// TwinCAT 3 PLC project Doble_Gato_PLC
// ProgramVersion: 3.1.4023.0
// libraries:
//   Tc2_Standard, * (Beckhoff Automation GmbH)
//   Tc2_System, * (Beckhoff Automation GmbH)
//   Tc2_Utilities, * (Beckhoff Automation GmbH)
//   Tc3_EventLogger, * (Beckhoff Automation GmbH)
//   Tc3_Module, * (Beckhoff Automation GmbH)
// project tree:
//   DUTs/ eBeltObject.TcDUT, eFeed.TcDUT, BeltStatus.TcDUT, OUTPUT_LABELS.TcDUT, INPUT_LABELS.TcDUT, U_IN_IO_Translate.TcDUT, U_OUT_IO_Translate.TcDUT
//   FBs/ FB_ButtonBox.TcPOU, FB_GatoPerro.TcPOU, FB_BeltControl.TcPOU
//   F/ F_TemperatureMethod.TcPOU
//   GVLs/ GENERAL.TcGVL
//   GVLs/IO/ IN.TcGVL, OUT.TcGVL
//   GVLs/SAFETY/ SAFETY.TcGVL
//   / PlcTask.TcTTO, SlowTask.TcTTO
//   POUs/ OVERVIEW_FBD.TcPOU, MAIN.TcPOU, P_Temperature_Obs.TcPOU, P_BACKGROUND.TcPOU, P_SAFETY.TcPOU, README.TcPOU
//   POUs/GENERAL/ P_WritePersistentData.TcPOU
// real-time tasks:
//   TASK PlcTask: cycle T#10ms, priority 20, ADS port 350
//   TASK SlowTask: cycle T#50000us, priority 30, ADS port 351
// I/O:
//   DEVICE Device 3 (EtherCAT Automation Protocol), AmsNetId 5.62.144.216.4.1
//   DEVICE Device 1 (EtherCAT), AmsNetId 5.62.144.216.2.1
//     Term 1 (EK1200) [EK1200-5000 EtherCAT Power supply (2A E-Bus)]
//       Term 2 (EL3204) [EL3204 4Ch. Ana. Input PT100 (RTD)]
//       Term 3 (EL1008) [EL1008 8Ch. Dig. Input 24V, 3ms]
//       Term 4 (EL2008) [EL2008 8Ch. Dig. Output 24V, 0.5A]
//       Term 5 (EL1809) [EL1809 16Ch. Dig. Input 24V, 3ms]
//       Term 6 (EL2809) [EL2809 16Ch. Dig. Output 24V, 0.5A]
//       Term 7 (EK1122) [EK1122 2 port EtherCAT junction]
//         Term 8 (EK1100) [EK1100 EtherCAT Coupler (2A E-Bus)]
//           Term 9 (EL1008) [EL1008 8Ch. Dig. Input 24V, 3ms]
//           Term 10 (EL2008) [EL2008 8Ch. Dig. Output 24V, 0.5A]
//           Term 11 (EL9011) [EL9011 End Terminal]
// variable links:
//   Doble Gato PLC/Doble Gato PLC Instance <-> Device 1 (EtherCAT)
//     SlowTask Inputs/GENERAL.EthercatDevState <-> Inputs/DevState
//     SlowTask Outputs/GENERAL.EthercatDevCtrl <-> Outputs/DevCtrl
//   Doble Gato PLC/Doble Gato PLC Instance <-> Device 1 (EtherCAT)/Term 1 (EK1200)/Term 2 (EL3204)
//     SlowTask Inputs/IN.ANALOG[{1..4}] <-> RTD Inputs Channel {1..4}/Value  (4 links)
//   Doble Gato PLC/Doble Gato PLC Instance <-> Device 1 (EtherCAT)/Term 1 (EK1200)/Term 3 (EL1008)
//     PlcTask Inputs/IN._DI/bArray[{1..8}] <-> Channel {1..8}/Input  (8 links)
//   Doble Gato PLC/Doble Gato PLC Instance <-> Device 1 (EtherCAT)/Term 1 (EK1200)/Term 4 (EL2008)
//     PlcTask Outputs/OUT._DO/bArray[{1..8}] <-> Channel {1..8}/Output  (8 links)
//   Doble Gato PLC/Doble Gato PLC Instance <-> Device 1 (EtherCAT)/Term 1 (EK1200)/Term 5 (EL1809)
//     PlcTask Inputs/IN._DI/bArray[{9..24}] <-> Channel {1..16}/Input  (16 links)
//   Doble Gato PLC/Doble Gato PLC Instance <-> Device 1 (EtherCAT)/Term 1 (EK1200)/Term 6 (EL2809)
//     PlcTask Outputs/OUT._DO/bArray[{9..24}] <-> Channel {1..16}/Output  (16 links)
//   Doble Gato PLC/Doble Gato PLC Instance <-> Device 1 (EtherCAT)/Term 1 (EK1200)/Term 7 (EK1122)/Term 8 (EK1100)/Term 10 (EL2008)
//     PlcTask Outputs/OUT._DO/bArray[{25..32}] <-> Channel {1..8}/Output  (8 links)
//   Doble Gato PLC/Doble Gato PLC Instance <-> Device 1 (EtherCAT)/Term 1 (EK1200)/Term 7 (EK1122)/Term 8 (EK1100)/Term 9 (EL1008)
//     PlcTask Inputs/IN._DI/bArray[{25..32}] <-> Channel {1..8}/Input  (8 links)
//   Doble Gato PLC/Doble Gato PLC Instance <-> Device 3 (EtherCAT Automation Protocol)
//     SlowTask Inputs/GENERAL.EthercatDev1 <-> Inputs/DevState

CONFIGURATION Doble_Gato_PLC
    RESOURCE PLC ON TwinCAT3
        TASK PlcTask(INTERVAL := T#10ms, PRIORITY := 20);
        TASK SlowTask(INTERVAL := T#50000us, PRIORITY := 30);
        PROGRAM MAIN WITH PlcTask : MAIN;
        PROGRAM P_Temperature_Obs WITH SlowTask : P_Temperature_Obs;
    END_RESOURCE
END_CONFIGURATION

// ---- DUTs/eBeltObject.TcDUT
{attribute 'qualified_only'}
{attribute 'strict'}
TYPE eBeltObject :
(
	EMPTY := 0,
	GATO := 1,
	PERRO := 2,
	MAGIC := 3
);
END_TYPE

// ---- DUTs/eFeed.TcDUT
{attribute 'qualified_only'}
{attribute 'to_string'}
TYPE eFeed :
(
	Stop := 0,
	Ready,
	Running,
	Fault,
	State4
);
END_TYPE

// ---- DUTs/BeltStatus.TcDUT
{attribute 'qualified_only'}
{attribute 'strict'}
TYPE BeltStatus :
(
	Idle := 0,
	Ready,
	Running,
	Error_status := 100

);
END_TYPE

// ---- DUTs/OUTPUT_LABELS.TcDUT
TYPE OUTPUT_LABELS :
STRUCT
//===== 	Box EL2008			
ButtonBox_Light	:		BOOL;
bOutput2		:		BOOL;
bOutput3		:		BOOL;
bOutput4		:		BOOL;
bOutput5		:		BOOL;
bOutput6		:		BOOL;
bOutput7		:		BOOL;
DoorSensor_Activator		:		BOOL;
//===== 	Box EL2809
bOutput9		:		BOOL;
bOutput10		:		BOOL;
bOutput11		:		BOOL;
bOutput12		:		BOOL;
bOutput13		:		BOOL;
bOutput14		:		BOOL;
bOutput15		:		BOOL;
bOutput16		:		BOOL;
bOutput17		:		BOOL;
bOutput18		:		BOOL;
bOutput19		:		BOOL;
bOutput20		:		BOOL;
bOutput21		:		BOOL;
bOutput22		:		BOOL;
bOutput23		:		BOOL;
bOutput24		:		BOOL;
//===== 	EK1100 EL2008
VFD_RUN_14			:		BOOL;
VFD_BACKWARD_15		:		BOOL;
VFD_FORWARD_16		:		BOOL;
LIGHT_White		:		BOOL;
LIGHT_Green		:		BOOL;
bOutput30		:		BOOL;
bOutput31		:		BOOL;
bOutput32		:		BOOL;

END_STRUCT
END_TYPE

// ---- DUTs/INPUT_LABELS.TcDUT
TYPE INPUT_LABELS :
STRUCT
//===== 	Box EL1008			
BTN_Feed		:		BOOL;
SWITCH_Right		:		BOOL;
SWITCH_Left		:		BOOL;
bInput4		:		BOOL;
bInput5		:		BOOL;
bInput6		:		BOOL;
bInput7		:		BOOL;
SM_Door_Sensor1		:		BOOL;
//===== 	Box EL1809
bInput9		:		BOOL;
SM_Wheel_RotationCount		:		BOOL;
bInput11		:		BOOL;
SL_Wheel_LightSensor1		:		BOOL;
bInput13		:		BOOL;
bInput14		:		BOOL;
bInput15		:		BOOL;
bInput16		:		BOOL;
bInput17		:		BOOL;
bInput18		:		BOOL;
bInput19		:		BOOL;
bInput20		:		BOOL;
bInput21		:		BOOL;
bInput22		:		BOOL;
bInput23		:		BOOL;
bInput24		:		BOOL;
//====		EL1100 -> EL1008
VFD_READY_20		:		BOOL;
bInput26		:		BOOL;
VFD_24		:		BOOL;
bInput28		:		BOOL;
VFD_26		:		BOOL;
bInput30		:		BOOL;
bInput31		:		BOOL;
SM_Gato_MagnetSensor		:		BOOL;

END_STRUCT
END_TYPE

// ---- DUTs/U_IN_IO_Translate.TcDUT
TYPE U_IN_IO_Translate :
UNION
	bArray :	ARRAY[1..32] OF BOOL;
	_Label :		INPUT_LABELS;
END_UNION
END_TYPE

// ---- DUTs/U_OUT_IO_Translate.TcDUT
TYPE U_OUT_IO_Translate :
UNION
	bArray :	ARRAY[1..32] OF BOOL;
	_Label :		OUTPUT_LABELS;
END_UNION
END_TYPE

// ---- GVLs/GENERAL.TcGVL
{attribute 'qualified_only'}
VAR_GLOBAL
	ReadyForAction		: BOOL;
	BlinkOn				: BOOL;
	BlinkFAST_On		: BOOL;
	BlinkSpecial_On		: BOOL;	
	Motor_OK			: BOOL;
	Manual				: BOOL;
	Auto				: BOOL;

// General information	
	sCelsius: STRING(16);
	sFahrenheit: STRING(16);
	sCosine: STRING(16);
	sKelvin: STRING(16);

	Gato : BOOL;
	Perro : BOOL;
	GatoCount: UINT;
	PerroCount: UINT;	
	
// Linked 'useless' variables to IO
	EthercatDevState 	AT%I*: UINT;
	Term2DevState 		AT%I*: UINT;
	EthercatDevCtrl 	AT%Q*: UINT;
	EthercatDev1		AT%I*: UINT;
	EthercatDev3		AT%I*: UINT;


END_VAR

// ---- GVLs/IO/IN.TcGVL
{attribute 'qualified_only'}
VAR_GLOBAL
	_DI				AT %I*: 	U_IN_IO_Translate;
	ANALOG			AT %I*:		ARRAY[1..4] OF INT;	// Temperature module
	
END_VAR

// ---- GVLs/IO/OUT.TcGVL
{attribute 'qualified_only'}
VAR_GLOBAL
	_DO 			AT%Q*:		U_OUT_IO_Translate;

END_VAR

// ---- GVLs/SAFETY/SAFETY.TcGVL
{attribute 'qualified_only'}
VAR_GLOBAL
	//Turvapiirien tilatiedot
	Safety_OK							AT%Q*	:BOOL;	//
	Doors_OK							AT%Q*	:BOOL;	//
	E_STOP_OK							AT%Q*	:BOOL;	//
	
END_VAR

// ---- POUs/MAIN.TcPOU
PROGRAM MAIN
VAR
	
END_VAR


P_Safety();						// Check doors, safety switches etc. before going through with main program

IF GENERAL.ReadyForAction AND SAFETY.Safety_OK THEN 	// If both signals indicating readyness are given, go through with main tasks.
		P_BACKGROUND();					// Background routines. Blinks etc
		P_WritePersistentData();		// Writes persistent variables to memory every 10 seconds
		OVERVIEW_FBD();					// FBD View of all FB's. Useful visualization of whats happening
			// P_Environment_Control 		-> Is a separate slow task, not to be called from MAIN
END_IF

END_PROGRAM

// ---- POUs/P_SAFETY.TcPOU
PROGRAM P_SAFETY
VAR
	Door1_Box	: BOOL;
	Door2_Fence : BOOL;
	Door3_Workbench : BOOL;
	
END_VAR


A_Doors();	// Checking if doors are open
A_Checks(); // Acting on sensor inputs

	//Virtual switches waiting for physical ones
	SAFETY.E_STOP_OK 		:= TRUE;
	GENERAL.Motor_OK		:= TRUE;
	
//============
// If VFD is ready and Security is satisfactory, global "Good To Go"-signal is given
IF GENERAL.Motor_OK AND SAFETY.Safety_OK THEN
	GENERAL.ReadyForAction := TRUE;
END_IF

ACTION A_Checks:
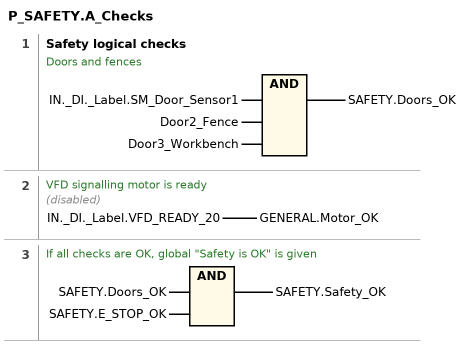
// NETWORK 1: Safety logical checks
// Doors and fences
SAFETY.Doors_OK := IN._DI._Label.SM_Door_Sensor1 AND Door2_Fence AND Door3_Workbench;

// NETWORK 2 (disabled)
// VFD signalling motor is ready
// GENERAL.Motor_OK := IN._DI._Label.VFD_READY_20;

// NETWORK 3
// If all checks are OK, global "Safety is OK" is given
SAFETY.Safety_OK := SAFETY.Doors_OK AND SAFETY.E_STOP_OK;
END_ACTION

ACTION A_Doors:
//"Door sensor" is active Output running to magnet sensor in door
OUT._DO._Label.DoorSensor_Activator := TRUE;

//========================

Door1_Box 		:= IN._DI._Label.SM_Door_Sensor1;	// Previously activated door sensor output is listened here
Door2_Fence 	:= TRUE;							// Not implemented physically	
Door3_Workbench := TRUE;							// Not implemented physically

IF (Door1_Box AND Door2_Fence AND Door3_Workbench) = TRUE THEN	// Checking through all doors and fences
	SAFETY.Doors_OK := TRUE;
	ELSE
		SAFETY.Doors_OK := FALSE;
END_IF
END_ACTION

END_PROGRAM

// ---- POUs/P_BACKGROUND.TcPOU
PROGRAM P_BACKGROUND
VAR
	bDoors : BOOL;
	State: INT;
	
	
//================	
	// Blink timer
	TIME_ON 			: TIME := T#1S;
	TIME_OFF 			: TIME := T#1S;	
	TIME_FAST_ON 		: TIME := T#250MS;
	TIME_FAST_OFF 		: TIME := T#250MS;
	TIME_SPECIAL_ON 	: TIME := T#50MS;
	TIME_SPECIAL_OFF 	: TIME := T#50MS;	
	
	BlinkTimer_ON: TON;
	BlinkTimer_OFF: TON;
	BlinkTimer_FAST_ON: TON;
	BlinkTimer_FAST_OFF: TON;
	BlinkTimer_SPEC_ON: TON;
	BlinkTimer_SPEC_OFF: TON;
	T_ON : BOOL;
	T_OFF : BOOL := TRUE;	
	T_FAST_ON : BOOL;
	T_FAST_OFF : BOOL := TRUE;	
	T_SPEC_ON : BOOL;
	T_SPEC_OFF : BOOL := TRUE;
//==================

	StateSpecial: INT;
	i: INT;
	Input1_RTRIG: R_TRIG;
	Input2_RTRIG: R_TRIG;
	tempCounter: INT;
	tempCounter2: INT;
	bSwitchToggle: BOOL;
END_VAR


//	A_ButtonBoxes();
//	A_FeedButton();
	Blink();
	Blink_Faster();
	Blink_Special();

ACTION A_Beacons:

END_ACTION

ACTION Blink:

BlinkTimer_ON(IN:= T_ON , PT:= TIME_ON , Q=> , ET=> );
IF BlinkTimer_ON.Q THEN
	T_ON 	:= GENERAL.BlinkOn:= FALSE;
	T_OFF 	:= TRUE;	
END_IF

BlinkTimer_OFF(IN:= T_OFF , PT:= TIME_OFF , Q=> , ET=> );
IF BlinkTimer_OFF.Q THEN
	T_ON 	:= GENERAL.BlinkOn := TRUE;
	T_OFF	:= FALSE;
END_IF
END_ACTION

ACTION Blink_Faster:


BlinkTimer_FAST_ON(IN:= T_FAST_ON , PT:= TIME_FAST_ON , Q=> , ET=> );
IF BlinkTimer_FAST_ON.Q THEN
	T_FAST_ON	:= GENERAL.BlinkFAST_On:= FALSE;
	T_FAST_OFF 	:= TRUE;	
END_IF

BlinkTimer_FAST_OFF(IN:= T_FAST_OFF , PT:= TIME_FAST_OFF , Q=> , ET=> );
IF BlinkTimer_FAST_OFF.Q THEN
	T_FAST_ON 	:= GENERAL.BlinkFAST_On := TRUE;
	T_FAST_OFF	:= FALSE;
END_IF
END_ACTION

ACTION Blink_Special:

CASE StateSpecial OF
0:

	IF i > 5 THEN
		StateSpecial := 1;
		i := 0;
		ELSE
		BlinkTimer_SPEC_ON(IN:= T_SPEC_ON , PT:= (TIME_SPECIAL_ON*5) , Q=> , ET=> );
		IF BlinkTimer_SPEC_ON.Q THEN
			T_SPEC_ON 	:= GENERAL.BlinkSpecial_ON:= FALSE;
			T_SPEC_OFF 	:= TRUE;	
		END_IF
		
		BlinkTimer_SPEC_OFF(IN:= T_SPEC_OFF , PT:= (TIME_SPECIAL_OFF*5) , Q=> , ET=> );
		IF BlinkTimer_SPEC_OFF.Q THEN
			T_SPEC_ON 	:= GENERAL.BlinkSpecial_ON := TRUE;
			T_SPEC_OFF	:= FALSE;
		i:= i+1;
		END_IF
	END_IF

	1: 

	IF i > 1 THEN
		StateSpecial := 0;
		i := 0;
		ELSE
		BlinkTimer_SPEC_ON(IN:= T_SPEC_ON , PT:= (TIME_SPECIAL_ON*10) , Q=> , ET=> );
		IF BlinkTimer_SPEC_ON.Q THEN
			T_SPEC_ON 	:= GENERAL.BlinkSpecial_ON:= FALSE;
			T_SPEC_OFF 	:= TRUE;	
		END_IF
		
		BlinkTimer_SPEC_OFF(IN:= T_SPEC_OFF , PT:= (TIME_SPECIAL_OFF*10) , Q=> , ET=> );
		IF BlinkTimer_SPEC_OFF.Q THEN
			T_SPEC_ON 	:= GENERAL.BlinkSpecial_ON := TRUE;
			T_SPEC_OFF	:= FALSE;
			i:= i+1;
		END_IF
	END_IF
END_CASE
END_ACTION

END_PROGRAM

// ---- POUs/GENERAL/P_WritePersistentData.TcPOU
PROGRAM P_WritePersistentData
VAR
	fbWritePersistentData: FB_WritePersistentData;
	StartTON: TON;
	iCounter: INT;

END_VAR

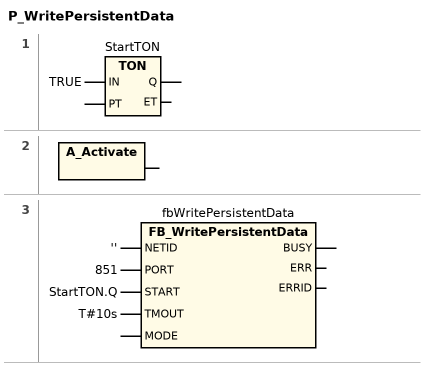
// NETWORK 1
StartTON(IN := TRUE); // TON

// NETWORK 2
A_Activate();

// NETWORK 3
fbWritePersistentData(NETID := '', PORT := 851, START := StartTON.Q, TMOUT := T#10s); // FB_WritePersistentData

ACTION A_Activate:

IF StartTON.Q THEN
	StartTON(IN := FALSE, PT:= T#1M);
		IF NOT fbWritePersistentData.BUSY THEN
		StartTON(IN := TRUE);
		iCounter := iCounter +1; IF iCounter > 50 THEN iCounter := 0; END_IF
		END_IF
END_IF
END_ACTION

END_PROGRAM

// ---- POUs/OVERVIEW_FBD.TcPOU
PROGRAM OVERVIEW_FBD
VAR
	fbButtonBox: FB_ButtonBox;
	fbBeltControl: FB_BeltControl;
	fbGatoPerro: FB_GatoPerro;
END_VAR

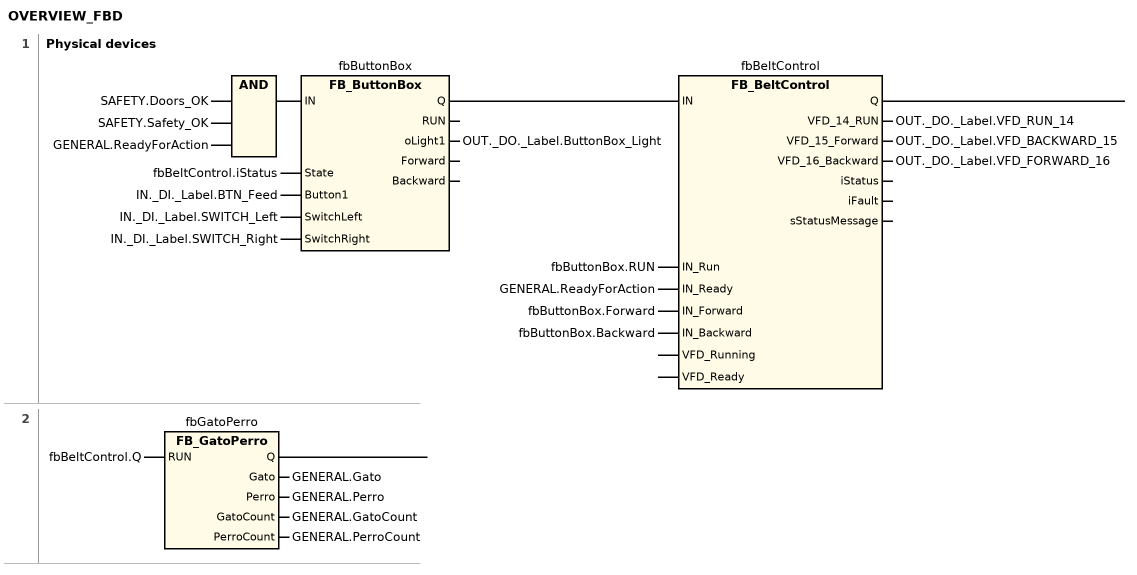
// NETWORK 1: Physical devices
fbButtonBox(
    IN := SAFETY.Doors_OK AND SAFETY.Safety_OK AND GENERAL.ReadyForAction,
    State := fbBeltControl.iStatus,
    Button1 := IN._DI._Label.BTN_Feed,
    SwitchLeft := IN._DI._Label.SWITCH_Left,
    SwitchRight := IN._DI._Label.SWITCH_Right,
    oLight1 => OUT._DO._Label.ButtonBox_Light); // FB_ButtonBox
fbBeltControl(
    IN := fbButtonBox.Q,
    IN_Run := fbButtonBox.RUN,
    IN_Ready := GENERAL.ReadyForAction,
    IN_Forward := fbButtonBox.Forward,
    IN_Backward := fbButtonBox.Backward,
    VFD_14_RUN => OUT._DO._Label.VFD_RUN_14,
    VFD_15_Forward => OUT._DO._Label.VFD_BACKWARD_15,
    VFD_16_Backward => OUT._DO._Label.VFD_FORWARD_16); // FB_BeltControl

// NETWORK 2
fbGatoPerro(
    RUN := fbBeltControl.Q,
    Gato => GENERAL.Gato,
    Perro => GENERAL.Perro,
    GatoCount => GENERAL.GatoCount,
    PerroCount => GENERAL.PerroCount); // FB_GatoPerro

END_PROGRAM

// ---- FBs/FB_ButtonBox.TcPOU
FUNCTION_BLOCK FB_ButtonBox
VAR_INPUT
	IN			: BOOL;
	State : 	(NOT_READY, ALL_READY, RUNNING, STOP, ERROR);	//Local ENUM
	Button1		: BOOL;
	SwitchLeft 	: BOOL;
	SwitchRight : BOOL;
END_VAR
VAR_OUTPUT
	Q 		: BOOL;
	RUN		: BOOL;
	oLight1 : BOOL;	
	Forward 	: BOOL;
	Backward 	: BOOL;
END_VAR
VAR
	BTN_Feed_TRIG: BOOL;
	Rtrig2: R_TRIG;
	Rtrig3: R_TRIG;
	tempCount1: INT;
	tempCount2: INT;
	tempCount3: INT;
	tempCount0: INT;

	RS1: RS;
	SwitchLeftRight_RS: BOOL;
	rTrig1: R_TRIG;
	RS_2: RS;
END_VAR

Q := IN;

// Button press handling
A_InputHandling();

// Button box light controls dictated by the state of Belt Control.
CASE State OF		// State is an input of 1-5 from BeltControl FB
	
	NOT_READY:
		oLight1 := FALSE;

	ALL_READY:
		oLight1 := GENERAL.BlinkOn;
		
	RUNNING:
		oLight1 := TRUE;		
		
	STOP:
		oLight1 := GENERAL.BlinkSpecial_On;

	ERROR:
		oLight1 := GENERAL.BlinkSpecial_On;
		
END_CASE

ACTION A_InputHandling:
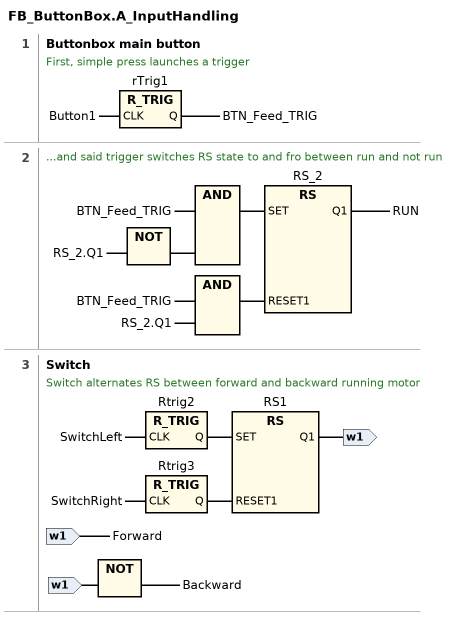
// NETWORK 1: Buttonbox main button
// First, simple press launches a trigger
rTrig1(CLK := Button1); // R_TRIG
BTN_Feed_TRIG := rTrig1.Q;

// NETWORK 2
// ...and said trigger switches RS state to and fro between run and not run
RS_2(SET := BTN_Feed_TRIG AND NOT RS_2.Q1, RESET1 := BTN_Feed_TRIG AND RS_2.Q1); // RS
RUN := RS_2.Q1;

// NETWORK 3: Switch
// Switch alternates RS between forward and backward running motor
Rtrig2(CLK := SwitchLeft); // R_TRIG
Rtrig3(CLK := SwitchRight); // R_TRIG
RS1(SET := Rtrig2.Q, RESET1 := Rtrig3.Q); // RS
Forward := RS1.Q1;
Backward := NOT RS1.Q1;
END_ACTION

END_FUNCTION_BLOCK

// ---- FBs/FB_BeltControl.TcPOU
FUNCTION_BLOCK FB_BeltControl
VAR_INPUT
	IN				: BOOL;
	IN_Run 			: BOOL; // Order to start running
	IN_Ready			: BOOL; // Safety ok, system ok, doors ok
	IN_Forward 			: BOOL;
	IN_Backward			: BOOL;
	VFD_Running		: BOOL;
	VFD_Ready		: BOOL;
	
END_VAR
VAR_OUTPUT
	Q : BOOL;
	VFD_14_RUN 	: BOOL;
	VFD_15_Forward		: BOOL;
	VFD_16_Backward		: BOOL;
	iStatus		: INT;
	iFault		: INT;
	sStatusMessage	: STRING;
END_VAR
VAR
	nMotorState: (NOT_READY, ALL_READY, RUNNING, STOP, ERROR);	//Local ENUM
	Stopping_TON: TON;
	sDirCase: (FORWARD, BACKWARD);
	Frw_Bck: INT;
	fbTcMessage: FB_TcMessage;	//Eventlogger messaging
		bIsInitialized : BOOL;
		bSendMessage : BOOL;
	
	iTempCounter: INT;
END_VAR

M_VariableChanges();
IF NOT IN_Ready THEN		// VFD signal of readiness. Simple way to work safely with VFD
	nMotorState :=0;
END_IF

CASE nMotorState OF
	NOT_READY:	
	sStatusMessage := 'Not ready. Stopped';
		IF IN_Ready THEN
		nMotorState := 1;	// When VFD signals it is ready, we can proceed
		END_IF

	ALL_READY:
	sStatusMessage := 'Ready to run. Motor Stopped';
		VFD_14_RUN := FALSE;
		VFD_15_Forward := FALSE;
		VFD_16_Backward := TRUE;
	
		IF IN_Run THEN		// Inputted signal from buttonbox or other remote to start
			nMotorState := 2;	// Move on to Running-state

			//Also send informational Eventlogger message:
			bIsInitialized := TRUE;
				IF bIsInitialized THEN
					bIsInitialized := FALSE;
					bSendMessage := TRUE;
					fbTcMessage.CreateEx(TC_Events.GatoPerroEvents.Start, 0);
				END_IF
			
		END_IF
		
	RUNNING:
							// Motor can either run forward or backward according to buttonbox switch
		CASE sDirCase  OF			
			BACKWARD:
				VFD_14_RUN := FALSE;
				VFD_15_Forward := TRUE;
				VFD_16_Backward := FALSE;
				sStatusMessage := 'Motor running: Backward';

			FORWARD:
				VFD_14_RUN := TRUE;
				VFD_15_Forward := FALSE;
				VFD_16_Backward := TRUE;
				sStatusMessage := 'Motor running: Forward';
		END_CASE

		IF NOT IN_Run THEN	
			nMotorState := 3;
		END_IF

	STOP:
		sStatusMessage := 'Stopping...';	// Motor is gradually stopped and slight delay is included before new start can be ordered
		VFD_14_RUN := FALSE;
		VFD_15_Forward := FALSE;
		VFD_16_Backward := TRUE;
		
		Stopping_TON(IN:=TRUE , PT:=T#2S , Q=> , ET=> );
			IF Stopping_TON.Q THEN
				Stopping_TON(IN:=FALSE);
				nMotorState := 0;
			END_IF
		
	ERROR:
		sStatusMessage := 'Error state';
	
		
END_CASE

A_Messaging();

ACTION A_Messaging:

//Sends tc eventlogger messages if it is primed previously

IF bSendMessage THEN
	bSendMessage := FALSE;
	iTempCounter := iTempCounter +1;
	fbTcMessage.Send(0);	// 0 = current timestamp
END_IF
END_ACTION

METHOD M_VariableChanges : BOOL
VAR_INPUT
END_VAR

IN 					:= Q;
VFD_15_Forward 		:= IN_Forward;
VFD_16_Backward 	:= IN_Backward;
iStatus 			:= nMotorState;
iFault 				:= 0;
Frw_Bck 			:= BOOL_TO_INT( IN_Forward);
sDirCase		 	:= Frw_Bck;
END_METHOD

END_FUNCTION_BLOCK

// ---- FBs/FB_GatoPerro.TcPOU
FUNCTION_BLOCK FB_GatoPerro
VAR_INPUT
	RUN 		: BOOL;
END_VAR
VAR_OUTPUT
	Q			: BOOL;
	Gato 		: BOOL;
	Perro 		: BOOL;
	GatoCount 	: UINT;
	PerroCount 	: UINT;

END_VAR
VAR
	R_TRIG_0: R_TRIG;
	R_TRIG_1: R_trig;
	GatoTrigger: BOOL;
	WheelLightTrigger: BOOL;
	R_TRIG_2: R_TRIG;
	RotationTrigger: BOOL;
	RotationCount: UINT;
	ObjectCount: UINT;
	GatoPrime: BOOL;
	bGato_or_Perro: BOOL;
	TON_PrimeDelay: TON;
	WheelTime1: TIME;
	WheelTime3: TIME;
	WheelTime2: TIME;
	GP_Check: UINT;
	//A_RotationMeasure VARs	
		tTimeNow: TIME;
		tRotationTime: TIME;
		tTimeStop: TIME;
		iRotations_In_Minute: DWORD;
		iTimenow: DWORD;
		iOneMinute: DWORD;
		iRotationTime: DWORD;
		iOne_Fourth_Rotations_Time: DWORD;
		iTenth_Of_Rotations_Time: DWORD;
		tOne_Fourth_Rotations_Time: TIME;
		tTenth_Of_Rotations_Time: TIME;
	tonLightSDelay: TON;
	ObjectDetectionTime: TIME := T#50MS;
	Prime_Start: BOOL;
END_VAR

Q := RUN;
A_SensorHandling();

// Rotation counter
IF RotationTrigger THEN
	RotationCount := RotationCount +1;

	// We need slight delay before Priming Gato. Perro could be just nearing the Light sensor and register as Gato
	// Lets calculate rotations per minute, divide it to 3/4th rotation and use these later on to prime Gato just in time
	A_RotationMeasure();
		tRotationTime;			// Informational
		iRotations_In_Minute;	// Informational		
END_IF

// Magnet sensor sees Gato
	// Lets add slight delay to avoid mixing with other object on wheel
	TON_PrimeDelay(IN:= Prime_Start, PT:= tOne_Fourth_Rotations_Time, Q=> , ET=> );
		IF GatoTrigger THEN
			Prime_Start := TRUE;
		END_IF
	// When timer is done, Gato is primed and will register in light sensor
		IF TON_PrimeDelay.Q THEN
			GatoPrime := TRUE;
			Prime_Start := FALSE;
		END_IF

// Light sensor sees an object
IF WheelLightTrigger THEN
	ObjectCount := ObjectCount +1;
	IF NOT GatoPrime THEN			// IF Gato is not primed, its Perro
		PerroCount := PerroCount +1;
		bGato_or_Perro := FALSE;
	ELSE							// If Gato is primed in previous steps, its Gato
		GatoPrime := FALSE;
		GatoCount := GatoCount +1;
		bGato_or_Perro := TRUE;
	END_IF

END_IF

// Which one was it
Gato 	:= bGato_or_Perro;
Perro 	:= NOT bGato_or_Perro;
// Finally, lit up a light for whichever object it was
A_SignalLights();

ACTION A_RotationMeasure:
// Calculate RPM from RotationTime, divide it to 1/4th rotation
// Also 1/10th rotation to filter light sensor input
// If rotation time is slowing too much, or stops, reset to 0.2s


// How long does one rotation take
	tTimeNow := TIME();
	tRotationTime := tTimeNow - tTimeStop;
	tTimeStop := tTimeNow;

//Some conversions:
	iTimenow := TIME_TO_DWORD(tTimeNow);
	iOneMinute := TIME_TO_DWORD(T#1M);
	iRotationTime := TIME_TO_DWORD(tRotationTime);

// Rotations_In_Minute
iRotations_In_Minute :=
	iOneMinute/iRotationTime;
	
// 1/4 and 1/10th rotation times
tOne_Fourth_Rotations_Time := DWORD_TO_TIME( iOne_Fourth_Rotations_Time :=
	iRotationTime/4);
tTenth_Of_Rotations_Time := DWORD_TO_TIME( iTenth_Of_Rotations_Time :=
	iRotationTime/10);
END_ACTION

ACTION A_SensorHandling:
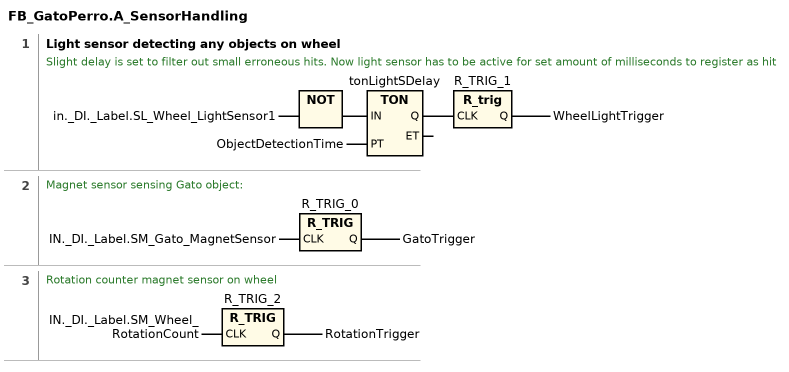
// NETWORK 1: Light sensor detecting any objects on wheel
// Slight delay is set to filter out small erroneous hits. Now light sensor has to be active for set amount of milliseconds to register as hit
tonLightSDelay(IN := NOT in._DI._Label.SL_Wheel_LightSensor1, PT := ObjectDetectionTime); // TON
R_TRIG_1(CLK := tonLightSDelay.Q); // R_trig
WheelLightTrigger := R_TRIG_1.Q;

// NETWORK 2
// Magnet sensor sensing Gato object:
R_TRIG_0(CLK := IN._DI._Label.SM_Gato_MagnetSensor); // R_TRIG
GatoTrigger := R_TRIG_0.Q;

// NETWORK 3
// Rotation counter magnet sensor on wheel
R_TRIG_2(CLK := IN._DI._Label.SM_Wheel_RotationCount); // R_TRIG
RotationTrigger := R_TRIG_2.Q;
END_ACTION

ACTION A_SignalLights:
// Lights signalling which object passed sensor
OUT._DO._Label.LIGHT_White := Gato;
OUT._DO._Label.LIGHT_Green := Perro;
END_ACTION

END_FUNCTION_BLOCK

// ---- POUs/P_Temperature_Obs.TcPOU
PROGRAM P_Temperature_Obs
VAR
	SA_BoxTemperature: REAL;
	rCelsius: REAL;

	rFahrenheit: REAL;
	rKelvin: REAL;
	rCosine: REAL;

END_VAR

// Analogue Temperature sensor inside box
SA_BoxTemperature := IN.ANALOG[1];
//=======================================

//Presenting conversions to display in HMI
F_TemperatureMethod(
	InputTemperature:= SA_BoxTemperature, 
	Celsius=> rCelsius, 
	Fahrenheit=> rFahrenheit, 
	Kelvin=> rKelvin,
	Cosine => rCosine);

// Turning temperature Reals to Global strings.
GENERAL.sCelsius := LREAL_TO_FMTSTR(in:= rCelsius, iPrecision:= 2, bRound:= 1);
GENERAL.sFahrenheit := LREAL_TO_FMTSTR(in:= rFahrenheit, iPrecision:= 2, bRound:= 1);
GENERAL.sKelvin := LREAL_TO_FMTSTR(in:= rKelvin, iPrecision:= 2, bRound:= 1);
GENERAL.sCosine := LREAL_TO_FMTSTR(in:= rCosine, iPrecision:= 5, bRound:= 1);

END_PROGRAM

// ---- F/F_TemperatureMethod.TcPOU
FUNCTION F_TemperatureMethod : REAL
VAR_INPUT
	InputTemperature:	REAL;
END_VAR
VAR_OUTPUT
	Celsius : 		REAL;
	Fahrenheit : 	REAL;
	Kelvin : 		REAL;
	Cosine :		REAL;
END_VAR
VAR
	K: REAL;
	C: REAL;
	F: REAL;
END_VAR

// Function handling analog temperature measurement 
C := InputTemperature/10; 
K := C + 273.15;
F := C * 1.8 +32;

Cosine		 	:= COS(C);
Celsius 		:= C;
Fahrenheit 		:= F;
Kelvin 			:= K;

END_FUNCTION

// ---- POUs/README.TcPOU
PROGRAM README
VAR
END_VAR

(*
//============
NAMING INPUTS USING UNION:
	Give Inputs/Outputs Specific Labels In: 
		DUT/INPUT_LABELS
		DUT/OUTPUT_LABELS
	
	Thus inputs have clear names and address:  
		IN._I._Label.Door_Sensor1
		
	IO is received into Array, and every input is then given a specific Label through Union. 
	IO can still be referenced in array form:
		IN._I.bArray[1];
	Because DUT/Union simply slaps a label on top of bArray[1..32], Door_Sensor1 and bArray[8] are the same thing and thus activate simultaneously.

//============
GATO E PERRO 
	Original idea of this demo project is to showcase and test different inputs, outputs and controls of PLC. Some features are needlessly complicated 
	considering the task, but are used for learning purposes. Several components are scavenged and repurposed, thus giving a but amateurish
	and hacky look to the project, but I still made an effort for professional finish.	

	Name is in Spanish to clearly distinguish test project from actual customer project. Future database names et al continue the same namoing
	convention to make it easier to copy/paste and change variables and names.
	
	End result of project is a cat figure running from dog figure, with magnetic and light sensor observing them.
	Distinguishing cat from a dog can be achieved in many ways, and I chose a middle ground between practicality, budget and reliability.
	Cat figure has a magnet glued behind it, thus "priming" the light sensor 
	-> next time a figure passes light sensor, its a cat. 
	-> If light sensor is not primed, its a dog.
	
	Inside the cabinet exists analog temperature sensor, a multiple port relay and green signal light.
 
	Cat and dog are running on electric motor, which is controlled by Vacon VFD.
	Due to availability, budget and preference, Vacon doesnt have any fancy input modules and is controlled with simple IO-pins. 
	Future learning potential is definitely there.

	 
=====================
	
	

*)

END_PROGRAM
